// TIA Portal V17 export
// export: Created 2024-01-30T08:49:14.1769563Z, ExportSetting WithDefaults, DisplayName Totally Integrated Automation Portal, DisplayVersion V17 Update 6, DisplayName TIA Portal Openness, DisplayVersion V17 Update 6, DisplayName TIA Portal Version Control Interface, DisplayVersion V17, DisplayName STEP 7 Professional, DisplayVersion V17 Update 6, DisplayName STEP 7 Safety, DisplayVersion V17 Update 6, DisplayName WinCC Advanced, DisplayVersion V17 Update 6
DATA_BLOCK "FESTO_CMMT_ST_DB"   // DB12
VERSION : 0.1
// stored: AutoNumber true, DBAccessibleFromOPCUA true, DBAccessibleFromWebserver true, InstanceOfName FESTO_CMMT_ST, InstanceOfType FB
"FESTO_CMMT_ST"
   // VAR
   //    Festo_PtP_Drives_PN_Instance { S7_SetPoint := 'True'} : "Festo_PtP_Drives_PN";
   // END_VAR
BEGIN
END_DATA_BLOCK
